FUNCTION F_ScaleToByteBeam : Byte
VAR_INPUT
	
	fActValue								:LREAL;
	fMaxValue								:LREAL;
	
END_VAR
VAR
	
	nValueBeam								:BYTE;
	
END_VAR
(* End *)

(* Scale to byte beam *)

	nValueBeam := TO_BYTE(TRUNC(F_Scaling(nAnalogIn:=TO_INT(ABS(fActValue)), fNumerator:=8.0, fDenominator:=fMaxValue )));
	
	CASE nValueBeam OF
		0	:	F_ScaleToByteBeam := 2#0;
		1	:	F_ScaleToByteBeam := 2#1;
		2	:	F_ScaleToByteBeam := 2#11;
		3	:	F_ScaleToByteBeam := 2#111;
		4	:	F_ScaleToByteBeam := 2#1111;
		5	:	F_ScaleToByteBeam := 2#11111;
		6	:	F_ScaleToByteBeam := 2#111111;
		7	:	F_ScaleToByteBeam := 2#1111111;
		8	:	F_ScaleToByteBeam := 2#11111111;
	END_CASE
	
(* End *)

END_FUNCTION

(* stored: Version 1.1.0.1, ProductVersion 3.1.4020.12
   POU F_ScaleToByteBeam: Id {a3bcd930-c52d-4ba1-a480-abe896caa435}, SpecialFunc None *)
